(* IEC 61131-3 sources: ConveyorControl-with-PLC/4E_Gruppe1_Graf_Projekt1/Class/HwControlBase, 1 file *)

(* ---- HwControlBase.st ---- *)
(*!
<Class
	Name               = "HwControlBase"
	Revision           = "1.10"
	RealtimeTask       = "false"
	CyclicTask         = "false"
	BackgroundTask     = "false"
	Sigmatek           = "true"
	OSInterface        = "false"
	HighPriority       = "false"
	Automatic          = "false"
	UpdateMode         = "Prescan"
	IconPath           = ".\Class\HwControl\HwControl.ico"
	SharedCommandTable = "true"
	Objectsize         = "(652,120)"
	Comment            = "Class to handle VaranManager and the cooperation with DiasMasterC&#13;&#10;BaseClass only contains empty implementation of UpdateRtPostScan">
	<Channels>
		<Server Name="Control" Visualized="true" Initialize="false" WriteProtected="true" Retentive="false" Comment="connect VaranManager classes"/>
		<Server Name="DiasMaster" Visualized="true" Initialize="false" WriteProtected="false" Retentive="false" Comment="connect to DiasMasterC Client if used (if Server is 1 class is connected)"/>
		<Server Name="State" Visualized="true" Initialize="false" WriteProtected="true" Retentive="false" Comment="state of HwControl class"/>
		<Client Name="RtDebug" Required="false" Internal="false" Comment="ATTENTION!!&#13;&#10;If client is activated hardware will be continue to work if a Realtime task is debugged.&#13;&#10;No Watchdog of hardware occures. RtPostScan will be called from RtPreScan which could lead to a different timing behaviour of the machine.&#13;&#10;&#13;&#10;(as Initvalue, default is off)"/>
		<Client Name="To_StdLib" Required="false" Internal="false"/>
		<Client Name="To_TaskObjectControl" Required="false" Internal="false" Comment="is automatically connected to OS class"/>
	</Channels>
	<Dependencies>
		<Files>
			<File Path=".\LSL_STITask.h" Include="false"/>
			<File Path=".\Class\VaranManager_Base\VaranManager_Base.h" Include="false"/>
		</Files>
	</Dependencies>
	<RevDoku>
		<Owner Company="Sigmatek" Author="BleErn"/>
		<Dokumentation Revision="1.10" Date="18.07.2013" Author="RamAnd" Company="Sigmatek" Description="Changed comment of RtDebug: Added warning, that the timing behaviour of the machine could be changed, when this client is set."/>
		<Dokumentation Revision="1.1" Date="27.02.2012" Author="RamAnd" Company="Sigmatek" Description="Added support for the SafetyManager"/>
		<Dokumentation Revision="1.0" Date="08.02.2010" Author="BleErn" Company="Sigmatek" Description="Creation of BaseClass for HwControl for implementation of HwRtPostScan"/>
	</RevDoku>
</Class>
*)
HwControlBase : CLASS
	TYPE
	  pVaranManager : ^VaranManager;
	  t_DMFunctions : STRUCT
	    p_RtFunction : pVoid;
	    p_SendSync : pVoid;
	    p_FinishIMProg : pVoid;
	    p_LastInit : pVoid;
	    p_This : pVoid;
	    sd_PllTime : DINT;
	    ud_DiasTime : UDINT;
	    sd_RtDebug : DINT;
	    sd_Reserved2 : DINT;
	    sd_Reserved3 : DINT;
	  END_STRUCT;
	  t_DiasMaster : STRUCT
	    ud_Counter : UDINT;
	    p_Functions : ^t_DMFunctions;
	  END_STRUCT;
	  t_VMFunctions : STRUCT
	    p_This : pVaranManager;
	    ud_VaranTime : UDINT;
	    b_IsAlsoClient : BOOL;
	    ud_SuperiorTime : UDINT;
	    b_HWClassSynchron : BOOL;
	    b_OverrideFrameCheck : BOOL;
	  END_STRUCT;
	  t_OneVaranManager : STRUCT
	    ud_Counter : UDINT;
	    ud_SuperiorSync : UDINT;
	    ud_SuperiorSyncActual : UDINT;
	    p_Functions : ^t_VMFunctions;
	  END_STRUCT;
	END_TYPE
  //Servers:
	Control 	: SvrChCmd_DINT;
	State 	: SvrCh_t_e_VaranErrors;
	DiasMaster 	: SvrCh_DINT;
  //Clients:
	To_TaskObjectControl 	: CltChCmd__TaskObjectControl;
	To_StdLib 	: CltChCmd__StdLib;
	RtDebug 	: CltCh_DINT;
  //Variables:
  //Functions:

	FUNCTION VIRTUAL GLOBAL UpdateRtPostScan;

	FUNCTION VIRTUAL GLOBAL AddSafetyManager
		VAR_INPUT
			pThis 	: pVirtualBase;
		END_VAR
		VAR_OUTPUT
			pFirstVM 	: pVirtualBase;
		END_VAR;

	FUNCTION VIRTUAL GLOBAL DisableSafetyManager;
  //Tables:
	FUNCTION @STD
		VAR_OUTPUT
			ret_code	: CONFSTATES;
		END_VAR;
	FUNCTION GLOBAL TAB @CT_;
END_CLASS;

#pragma usingLtd _StdLib
#pragma usingLtd _TaskObjectControl

#pragma usingLtd VaranManager

FUNCTION VIRTUAL GLOBAL HwControlBase::UpdateRtPostScan

END_FUNCTION

#pragma warning(disable: 73)
#pragma warning(disable: 76)
FUNCTION VIRTUAL GLOBAL HwControlBase::AddSafetyManager
	VAR_INPUT
		pThis 	: pVirtualBase;
	END_VAR
	VAR_OUTPUT
		pFirstVM 	: pVirtualBase;
	END_VAR

END_FUNCTION
#pragma warning(default: 73)
#pragma warning(default: 76)

FUNCTION VIRTUAL GLOBAL HwControlBase::DisableSafetyManager

END_FUNCTION
